Fanuc KAREL source: kx00009.KL

-- PROVISIONAL review KL for V770-1; original PC SHA256 41b5b66439cad3d75a1b1bb107d7115b3205900b7475acca83e69a6342fffc2e
-- Incomplete behavior may be omitted. Consult companion uncertainty JSON. Do not deploy.
PROGRAM KX00009
%NOLOCKGROUP
VAR
  I : INTEGER
  J : INTEGER
  B : BOOLEAN
  F : FILE
  S : STRING[80]
-- UNRESOLVED_DECL P type=000102
BEGIN
  -- UNRESOLVED_PC offsets 5-7; opcodes 9C,4F
  -- UNRESOLVED_PC offsets 12-16; opcodes 7F
END KX00009
